// TIA Portal V19 export
DATA_BLOCK "A0303_Sollevamento_PERS"   // DB105
// stored: MemoryReserve 100
   VAR RETAIN
      Par : Struct
         Ax_Man : "Positioning_DOL_Machine_Par";
         Ax_Testa_Pers { ExternalAccessible := 'False'; ExternalVisible := 'False'; ExternalWritable := 'False'} : "Positioning_DOL_Machine_Pers_Data";
         Ax_Coda_Pers { ExternalAccessible := 'False'; ExternalVisible := 'False'; ExternalWritable := 'False'} : "Positioning_DOL_Machine_Pers_Data";
         Enc : Struct
            Testa : "PosFbk_RTN";
            Coda { S7_SetPoint := 'True'} : "PosFbk_RTN";
         END_STRUCT;
      END_STRUCT;
      Par_Mach : Struct
         PosDeposito : LReal := 515.0;
         OffsetPrelievo : LReal := 25.0;
         ToleranceWindow : LReal := 1.0;
      END_STRUCT;
   END_VAR
BEGIN
   Par.Ax_Man.PosTolerance := 0.5;
   Par.Ax_Man.Minus_Limit := 5.0;
   Par.Ax_Man.Plus_Limit := 518.0;
   Par.Ax_Man.PreCutOff := 0.2;
   Par.Ax_Man.PreEndLowSpeed := 5.0;
   Par.Ax_Man.PreEndMedSpeed := 10.0;
   Par.Ax_Man.LowSpeed := 5.0;
   Par.Ax_Man.MedSpeed := 60.0;
   Par.Ax_Man.HighSpeed := 90.0;
   Par.Ax_Man.Man_Speed := 100.0;
   Par.Ax_Testa_Pers.AxisHomed := TRUE;
   Par.Ax_Coda_Pers.AxisHomed := TRUE;
   Par.Enc.Testa.Preset.Pulses := 1_524_110_052;
   Par.Enc.Testa.Preset.Units := 8.0;
   Par.Enc.Testa.Config.Resolution := 1.3435752;
   Par.Enc.Coda.Preset.Pulses := 965_337_904;
   Par.Enc.Coda.Preset.Units := 5.0;
   Par.Enc.Coda.Config.Resolution := 1.3435752;
END_DATA_BLOCK
